INTERFACE ITwoPointMovement

PROPERTY InHomePos : BOOL
GET
END_GET
END_PROPERTY

PROPERTY InWorkPos : BOOL
GET
END_GET
END_PROPERTY

METHOD ToHomePos : BOOL
VAR_INPUT
END_VAR
END_METHOD

METHOD ToWorkPos : BOOL
VAR_INPUT
END_VAR
END_METHOD

END_INTERFACE

(* stored: Version 1.1.0.1, ProductVersion 3.1.4024.11
   Itf ITwoPointMovement: Id {394d3116-9955-4ae0-a2f6-ebc87ee1b0c5}
   Property InHomePos: Id {b024296b-3083-44b9-af98-8d049e4d34ce}
   Get Get: Id {8c62b914-370b-435a-9a73-e3d4191f4dac}
   Property InWorkPos: Id {efd760dc-ecda-4694-b4e3-511f93d9e477}
   Get Get: Id {0d80be22-29fd-446d-86e5-298a039b24a1}
   Method ToHomePos: Id {44928774-89d8-46ee-92f2-8cee959caa80}
   Method ToWorkPos: Id {6ae4c225-7cf1-497c-b851-8282c53f8fa0} *)
